{attribute 'GeneratedUsingTerminal: AES-D-BC-ECAT Gen2-0001'}
{attribute addProperty BoxType "AES-D-BC-ECAT Gen2-0001"}
{attribute addProperty Id "Web_App_DisableAT %Q*BOOL1Freeze_OutputAT %Q*BOOL1HL_SwapAT %Q*BOOL1Default_Modul_ControlAT %Q*BOOL1"}
{attribute addProperty CRC "1649935978"}
{attribute addProperty Size "4"}
TYPE Device_Control_6258066A EXTENDS TcoIo.OutputBase_10CEE7DE :
STRUCT
	{attribute addProperty Name "Web_App_Disable"}
	Web_App_Disable AT %Q* : BOOL;
	{attribute addProperty Name "Freeze_Output"}
	Freeze_Output AT %Q* : BOOL;
	{attribute addProperty Name "HL_Swap"}
	HL_Swap AT %Q* : BOOL;
	{attribute addProperty Name "Default_Modul_Control"}
	Default_Modul_Control AT %Q* : BOOL;
END_STRUCT
END_TYPE

(* stored: Version 1.2.0.0
   DUT Device_Control_6258066A: Id {a457fb2e-6030-480c-98b0-0847672f08e9} *)
